// TIA Portal V19 export
VAR_GLOBAL   // PLC tag table "LB131"
   LB131_Decoiler_Lp_Bwd AT %Q118.5 : Bool;   // 332SH2
   LB131_Decoiler_Lp_Fwd AT %Q118.4 : Bool;   // 332SH1
   LB131_Decoiler_Pb_Bwd AT %I121.6 : Bool;   // 332SH2
   LB131_Decoiler_Pb_Fwd AT %I121.5 : Bool;   // 332SH1
   LB131_Peeler_Lp_Bwd AT %Q119.3 : Bool;   // 333SH2
   LB131_Peeler_Lp_Down AT %Q119.5 : Bool;   // 333SH4
   LB131_Peeler_Lp_Fwd AT %Q119.2 : Bool;   // 333SH1
   LB131_Peeler_Lp_Up AT %Q119.4 : Bool;   // 333SH3
   LB131_Peeler_Pb_Bwd AT %I122.4 : Bool;   // 333SH2
   LB131_Peeler_Pb_Down AT %I122.6 : Bool;   // 333SH4
   LB131_Peeler_Pb_Fwd AT %I122.3 : Bool;   // 333SH1
   LB131_Peeler_Pb_Up AT %I122.5 : Bool;   // 333SH3
   LB131_Snubber_Lp_Bwd AT %Q119.1 : Bool;   // 332SH6
   LB131_Snubber_Lp_Down AT %Q118.7 : Bool;   // 332SH4
   LB131_Snubber_Lp_Fwd AT %Q119.0 : Bool;   // 332SH5
   LB131_Snubber_Lp_Up AT %Q118.6 : Bool;   // 332SH3
   LB131_Snubber_Pb_Bwd AT %I122.2 : Bool;   // 332SH6
   LB131_Snubber_Pb_Down AT %I122.0 : Bool;   // 332SH4
   LB131_Snubber_Pb_Fwd AT %I122.1 : Bool;   // 332SH5
   LB131_Snubber_Pb_Up AT %I121.7 : Bool;   // 332SH3
   LB131_Straighetner_Lp_Bwd AT %Q119.7 : Bool;   // 333SH6
   LB131_Straighetner_Lp_Fwd AT %Q119.6 : Bool;   // 333SH5
   LB131_Straightener_Lift_Pb_Close AT %I123.0 : Bool;   // 333SA1
   LB131_Straightener_Lift_Pb_Open AT %I122.7 : Bool;   // 333SA1
   LB131_Straightener_Pb_Bwd AT %I123.2 : Bool;   // 333SH6
   LB131_Straightener_Pb_Fwd AT %I123.1 : Bool;   // 333SH5
   LB131_Button_R AT %I1034.4 : Bool;   // 104DI4 - 199SB2
   LB131_Button_L AT %I1034.0 : Bool;   // 104DI0 - 199SB1
END_VAR
